// TIA Portal V19 export
TYPE "LAF_typeAxisDiagStatusSensor"
TITLE = LAF_typeAxisDiagStatusSensor
// Status and actual values of all encoders of a Technology Object
// stored: Access Published
   STRUCT
      operativeSensor { ExternalWritable := 'False'} : UDInt := 1;   // Operative sensor/encoder
      sensor { ExternalWritable := 'False'} : Array[1..4] of "LAF_typeAxisDiagSensor";
   END_STRUCT;
END_TYPE
